FUNCTION_BLOCK FB_Temp_Sensor
VAR_INPUT
END_VAR
VAR_OUTPUT
	temp_out : REAL;
	temp_in AT %I* : INT;
END_VAR
VAR
	sensorlimit_high : REAL := 90.0;
	sensorlimit_low : REAL := -30.0;
END_VAR

// conversion from Bit value to temperature. 0 ~ -30 °C, 32767 ~ 90 °C
temp_out := (INT_TO_REAL(temp_in) / 32767 * (sensorlimit_high - sensorlimit_low)) + sensorlimit_low;

END_FUNCTION_BLOCK

(* stored: Version 1.1.0.1, ProductVersion 3.1.4024.9
   POU FB_Temp_Sensor: Id {5862196d-9579-4df5-99e3-f378128664c6}, SpecialFunc None *)
